// TIA Portal V17 export
// export: Created 2026-07-06T15:33:03.5629616Z, ExportSetting WithDefaults, DisplayName Totally Integrated Automation Portal, DisplayVersion V17, DisplayName TIA Portal Openness, DisplayVersion V17, DisplayName TIA Portal Version Control Interface, DisplayVersion V17, DisplayName STEP 7 Professional, DisplayVersion V17, DisplayName STEP 7 Safety, DisplayVersion V17, DisplayName WinCC Professional, DisplayVersion V17
DATA_BLOCK "kinco_BMS_TRCV_DB"   // DB8
// stored: AutoNumber true, DBAccessibleFromOPCUA true, InstanceOfName TRCV, OfSystemLibElement TRCV, OfSystemLibVersion 4.0
"TRCV"
   // VAR_INPUT
   //    EN_R : Bool;
   //    ID : CONN_OUC;
   //    LEN : UDInt;
   //    ADHOC : Bool;
   // END_VAR
   // VAR_OUTPUT
   //    NDR : Bool;
   //    BUSY : Bool;
   //    ERROR : Bool;
   //    STATUS : Word;
   //    RCVD_LEN : UDInt;
   // END_VAR
   // VAR_IN_OUT
   //    DATA : Variant;
   //    ADDR : Variant;
   // END_VAR
BEGIN
END_DATA_BLOCK
